Staubli VAL3: onF8Event.pgx

program onF8Event(bool& x_bExit[])
  local string l_sMessage
  local string l_sButton[2]
  local num l_nIndex
  local string l_sEvent
  local num l_nKey
  local string l_sItem
begin
  // look if the bButton is enable
  if bButton[7]
    //
    // EXIT or change Session
    //
    if saveData:bMultiSession and saveData:mode>=1
      // init
      use:nView=0
      // ask to change session or quit valplast
      call use:clear(0,13)
      call use:typeMenu(8,"<-")
      call use:setSizeList(30,9,8,2)
      call use:listcreate("")
      l_sItem="Quit"
      call use:listadd(l_sItem)
      l_sItem="Session"
      call use:listadd(l_sItem)
      call use:listupdate(0)
      // loop for a response
      do
        // read a key
        l_nKey=get()
        call use:listevent(l_nKey,l_nIndex,l_sEvent)
      until l_nKey==255 or l_nKey==270
      //
      if l_nKey!=255
        switch l_nIndex
          case 0
            //quit
            // clear the screen
            cls()
            // ask if the user want change the sesion
            call language:message(l_sMessage,4)
            // get the yes_no button Key
            call language:getYesNo(l_sButton)
            // ask the question
            call use:yes_no(l_sMessage,l_sButton,x_bExit)
          break
          case 1
            // change session
            call changeSession()
          break
        endSwitch
      endIf
    elseIf saveData:bMultiSession and saveData:mode==0
      call changeSession()
    else
      // ask if the user want change the sesion
      call language:message(l_sMessage,4)
      // get the yes_no button Key
      call language:getYesNo(l_sButton)
      // ask the question
      call use:yes_no(l_sMessage,l_sButton,x_bExit)
    endIf
  endIf
end
